type ST_Syntax_Mini : struct nId     : int; bActive : bool; sName   : string(32); end_struct end_type

(* stored: Version 1.1.0.1, ProductVersion 3.1.4024.16
   DUT ST_Syntax_Mini: Id {b4e196bd-4e4f-43f2-bf0d-fce6511685f0} *)
